// This function has been automatically generated from the project information.
{attribute 'signature_flag' := '1073741824'}
{attribute 'TcGenerated'}
{attribute 'no-analysis'}
FUNCTION F_GetCompany : WSTRING
VAR_INPUT
	
END_VAR

F_GetCompany := "FisoThemes";

END_FUNCTION

(* stored: Version 1.1.0.1
   POU F_GetCompany: Id {15314c0a-f8e3-0d42-1bcc-e8eb68224425}, SpecialFunc None *)
